{attribute 'qualified_only'}
VAR_GLOBAL
	stKrajalnica							: DUT_Krajalnica_Parametry;
END_VAR

(* stored: Version 1.1.0.1, ProductVersion 3.1.4024.11
   GVL GVL_Parametry: Id {a710716c-0c46-49ed-bfcd-a6b5c3064ce3} *)
